// TIA Portal V16 export
// export: Created 2022-08-08T12:29:18.6431506Z, ExportSetting WithDefaults, DisplayName Totally Integrated Automation Portal, DisplayVersion V16, DisplayName TIA Portal Version Control Interface, DisplayVersion V16, DisplayName TIA Portal Openness, DisplayVersion V16, DisplayName SINAMICS Startdrive Advanced, DisplayVersion V16, DisplayName SINAMICS Startdrive G130, G150, S120, S150, SINAMICS MV, S210, DisplayVersion V16, DisplayName SINAMICS Startdrive G110M, G120, G120C, G120D, G120P, DisplayVersion V16, DisplayName STEP 7 Professional, DisplayVersion V16, DisplayName STEP 7 Safety, DisplayVersion V16, DisplayName WinCC Professional, DisplayVersion V16
VAR_GLOBAL   // PLC tag table "Automatic_Gate_Example"
   stop AT %I0.0 : Bool;
   overcurrent_relay AT %I0.1 : Bool;
   system AT %M0.0 : Bool;
   up_directon_sensor AT %I0.5 : Bool;
   down_direction_sensor AT %I0.4 : Bool;
   open_limit AT %I0.2 : Bool;
   close_limit AT %I0.3 : Bool;
   open_gate AT %Q0.0 : Bool;
   close_gate AT %Q0.1 : Bool;
   gate_time AT %M0.1 : Bool;
END_VAR
